(* IEC 61131-3 sources: CODESYS-IO-Visualization/CODESYS-IO-Visualization.fbsproj/Subs/Misc, 3 files *)

(* ---- BitCount.prg.st ---- *)
PROGRAM BitCount

VAR_INPUT
	value: DWORD;
END_VAR

VAR_OUTPUT
	Count: INT;
END_VAR

WHILE value > 0 DO
	IF (value.0) THEN
		Count := Count + 1;
	END_IF;
	value := SHR(value,1);
END_WHILE;

(* ---- Random.prg.st ---- *)
PROGRAM Random

VAR_IN_OUT
	value: REAL;
END_VAR

VAR
	last: REAL;
	time_ms: DWORD;
	time_ms2: DWORD;
	timeBitsOn: INT;
	timeBitsOn2: INT;
END_VAR

last := value;
time_ms := TIME_TO_DWORD(TIME());

BitCount(value := time_ms, Count => timeBitsOn);

time_ms.31 := time_ms.2;
time_ms.30 := time_ms.5;
time_ms.29 := time_ms.4;
time_ms.27 := time_ms.0;
time_ms.26 := time_ms.7;
time_ms.25 := time_ms.6;
time_ms.24 := time_ms.3;

BitCount(value := time_ms, Count => timeBitsOn2);

time_ms := ROL(time_ms,timeBitsOn2) OR 16#80000001;
time_ms := time_ms MOD 71474513 + INT_TO_DWORD(timeBitsOn + 77);
value := DWORD_TO_REAL(time_ms) / 10000000.0 * (2.71828182845904523536028747135266249 - LIMIT(0.0,last,1.0));
value := ABS(value - DINT_TO_REAL(REAL_TO_DINT(value)));

(* ---- ValueRamp.prg.st ---- *)
PROGRAM ValueRamp

VAR_IN_OUT
	value: ValueRamp_UDT;
END_VAR

VAR
	DBMin: REAL;
	DBMax: REAL;
	DoRamp: BOOL;
END_VAR

CycleTime(value := value.CT);

IF (value.CT.mSec = 0) THEN
	RETURN;
END_IF;

DBMin := value.In - value.DB;
DBMax := value.In + value.DB;

DoRamp := TRUE;

IF (value.Track) THEN
	DoRamp := FALSE;
END_IF;

IF (value.Out > DBMin) AND (value.Out < DBMax) THEN
	DoRamp := FALSE;
END_IF;

IF (NOT value.Disable) THEN
	IF (DoRamp) THEN
		IF (value.Out < value.In) THEN
			value.Out := value.Out + (ABS(value.Rate) * value.CT.Sec);
		ELSE
			value.Out := value.Out - (ABS(value.Rate) * value.CT.Sec);
		END_IF;
	ELSE
		value.Out := value.In;
	END_IF;
END_IF;

value.Err := value.Out - value.In;

IF (value.Err > 0.0) THEN
	value.Status := ValueRampStatus_ENUM.OutHigh;
ELSIF (value.Err < 0.0) THEN
	value.Status := ValueRampStatus_ENUM.OutLow;
ELSE
	value.Status := ValueRampStatus_ENUM.Matched;
END_IF;
